ABB RAPID module: ReadTextMoveColor.mod

MODULE ReadTextMoveV2
    !   This module reads text from the target .txt file and moves to the points contained therein.
    !   Joshua Crook CM 1601   1-29-2016.
    VAR iodev pointsFile;
    PERS num paintHeight:=10;
    PERS num canvasHeight:=0;
    PERS num PAINT_MAX_DIST:=50;
    ! The largest usable square area the robot can draw in is 500mm wide by 150mm tall
    ! This is a rectangular large canvas, about 19.6" by 9.8"
    PERS num canvasXmin:=400;
    PERS num canvasXmax:=650;
    PERS num canvasYmin:=-250;
    PERS num canvasYmax:=250;

    VAR num sizeX;
    VAR num sizeY;
    VAR string tempStr;
    VAR num tempSF;
    VAR bool sizePassed:=FALSE;

    VAR num XTGT:=0;
    ! X target
    VAR num YTGT:=0;
    ! Y Target

    VAR num lastX:=0;
    VAR num lastY:=0;

    VAR string STRX;
    VAR string STRY;
    VAR string STRColor;
    VAR string lastColor:="A";
    !Arbitrary initialization value.

    VAR bool okX;
    VAR bool okY;
    VAR bool Skip;

    VAR num vX;
    VAR num vY;

    VAR num angleX;
    VAR num angleY;
    !measured in degrees from vertical.
    VAR num brushAngle:=10;

    VAR num vectorMag;
    VAR num distanceTravelled;

    PERS robtarget overA;
    PERS robtarget colorA;

    PERS robtarget overB;
    PERS robtarget colorB;

    PERS robtarget overC;
    PERS robtarget colorC;

    PERS robtarget overD;
    PERS robtarget colorD;

    PERS robtarget overE;
    PERS robtarget colorE;

    PERS robtarget overF;
    PERS robtarget colorF;

    PERS robtarget overClean;
    PERS robtarget clean;

    VAR num CaseHit;


    VAR orient ZeroZeroQuat:=[0.7071067811,0,0.7071067811,0];
    !vertical for paint can, etc.
    VAR orient paintStrokeQuat:=[0.7071067811,0,0.7071067811,0];
    !will change according to paintstroke vector.
    PERS num SF:=0.5;
    PERS num brushLength:=200;
    PERS num XOffset:=260;
    PERS num YOffset:=-150;
    PERS tooldata paintBrush:=[TRUE,[[87,0,146],[1,0,0,0]],[0.2,[0,0,146],[0,0,1,0],0,0,0]];

    PROC main()
        initializeColors;
        Open "HOME:/dumbSquare.txt",pointsFile\Read;
        distanceTravelled:=0;
        readSize;
        IF sizePassed=TRUE THEN
            readCoords;
            GotoPaint(STRColor);
            !first dip
            WHILE okX AND okY DO
                ! While we have data points in the file.
                moveToXY XTGT,YTGT;
                readCoords;
            ENDWHILE

        ENDIF

        Close pointsFile;
        ! exit.
    ENDPROC

    PROC initializeColors()
        overA:=[[514+brushLength,75,paintHeight+50],ZeroZeroQuat,[0,0,0,0],[9E9,9E9,9E9,9E9,9E9,9E9]];
        colorA:=[[514+brushLength,75,paintHeight],ZeroZeroQuat,[0,0,0,0],[9E9,9E9,9E9,9E9,9E9,9E9]];

        overB:=[[514+brushLength,50,paintHeight+50],ZeroZeroQuat,[0,0,0,0],[9E9,9E9,9E9,9E9,9E9,9E9]];
        colorB:=[[514+brushLength,50,paintHeight],ZeroZeroQuat,[0,0,0,0],[9E9,9E9,9E9,9E9,9E9,9E9]];

        overC:=[[514+brushLength,25,paintHeight+50],ZeroZeroQuat,[0,0,0,0],[9E9,9E9,9E9,9E9,9E9,9E9]];
        colorC:=[[514+brushLength,25,paintHeight],ZeroZeroQuat,[0,0,0,0],[9E9,9E9,9E9,9E9,9E9,9E9]];

        overD:=[[514+brushLength,0,paintHeight+50],ZeroZeroQuat,[0,0,0,0],[9E9,9E9,9E9,9E9,9E9,9E9]];
        colorD:=[[514+brushLength,0,paintHeight],ZeroZeroQuat,[0,0,0,0],[9E9,9E9,9E9,9E9,9E9,9E9]];

        overE:=[[514+brushLength,-25,paintHeight+50],ZeroZeroQuat,[0,0,0,0],[9E9,9E9,9E9,9E9,9E9,9E9]];
        colorE:=[[514+brushLength,-25,paintHeight],ZeroZeroQuat,[0,0,0,0],[9E9,9E9,9E9,9E9,9E9,9E9]];

        overF:=[[514+brushLength,-50,paintHeight+50],ZeroZeroQuat,[0,0,0,0],[9E9,9E9,9E9,9E9,9E9,9E9]];
        colorF:=[[514+brushLength,-50,paintHeight],ZeroZeroQuat,[0,0,0,0],[9E9,9E9,9E9,9E9,9E9,9E9]];

        overClean:=[[514+brushLength,-50,paintHeight+50],ZeroZeroQuat,[0,0,0,0],[9E9,9E9,9E9,9E9,9E9,9E9]];
        clean:=[[514+brushLength,-50,paintHeight],ZeroZeroQuat,[0,0,0,0],[9E9,9E9,9E9,9E9,9E9,9E9]];

    ENDPROC

    ! Reads the size off the passed file
    PROC readSize()
        sizePassed:=FALSE;
        ! This should be the X-size
        tempStr:=ReadStr(pointsFile\Delim:=",");
        okX:=StrToVal(tempStr,sizeX);
        ! This should be the Y-size
        tempStr:=ReadStr(pointsFile\Delim:=",");
        okY:=StrToVal(tempStr,sizeY);
        ! This should be a ';'
        tempStr:=ReadStr(pointsFile\Delim:=",");
        IF tempStr=";" THEN
            sizePassed:=TRUE;
            ! are we over the size constraints and in need of a scaling factor?
            IF (sizeX>(canvasXmax-canvasXmin)) OR (sizeY>(canvasYmax-canvasYmin)) THEN
                ! the Y proportion should be the scaling factor, as it was the smaller number
                IF ((canvasXmax-canvasXmin)/sizeX)>((canvasYmax-canvasYmin)/sizeY) THEN
                    SF:=(canvasYmax-canvasYmin)/sizeY;
                ELSE
                    SF:=(canvasXmax-canvasXmin)/sizeX;
                ENDIF

            ENDIF

        ELSE
            ErrLog 4800,"Data Error","The canvas size data was malformed","","","";
        ENDIF

    ENDPROC


    !   Reads the text file.
    PROC readCoords()
        STRX:=ReadStr(pointsFile\Delim:=",");
        okX:=StrToVal(STRX,XTGT);
        !End of a line.
        IF STRX=";" THEN
            STRColor:=ReadStr(pointsFile\Delim:=",");
            ! read the X value of the first point in the new line.
            STRX:=ReadStr(pointsFile\Delim:=",");
            STRY:=ReadStr(pointsFile\Delim:=",");

            okX:=StrToVal(STRX,XTGT);
            okY:=StrToVal(STRY,YTGT);

            checkForBadPoints XTGT,YTGT;

            XTGT:=(SF*XTGT)+canvasXmin;
            YTGT:=(SF*YTGT)+canvasYmin;
            CaseHit:=0;

        ELSEIF okX=FALSE THEN
            !Beginning of a file.
            STRColor:=STRX;
            STRX:=ReadStr(pointsFile\Delim:=",");
            STRY:=ReadStr(pointsFile\Delim:=",");

            okX:=StrToVal(STRX,XTGT);
            okY:=StrToVal(STRY,YTGT);

            checkForBadPoints XTGT,YTGT;

            XTGT:=(SF*XTGT)+canvasXmin;
            YTGT:=(SF*YTGT)+canvasYmin;
            lastX:=XTGT;
            lastY:=YTGT;
            CaseHit:=1;

        ELSEIF okX=TRUE THEN

            !we've already read the X value and it's not a character for a new line to be drawn.
            STRY:=ReadStr(pointsFile\Delim:=",");
            okY:=StrToVal(STRY,YTGT);

            checkForBadPoints XTGT,YTGT;

            XTGT:=(SF*XTGT)+canvasXmin;
            YTGT:=(SF*YTGT)+canvasYmin;
            CaseHit:=2;

        ENDIF
        !end of a file.
        IF (NOT okX) AND (NOT okY) THEN
            MoveL [[LastX,LastY,canvasHeight+30],ZeroZeroQuat,[0,0,0,0],[9E9,9E9,9E9,9E9,9E9,9E9]],v500,z0,paintBrush;
            MoveL overA,v500,fine,paintBrush;
        ENDIF
    ENDPROC

    ! Halts the robot if we get bad points.
    PROC checkForBadPoints(num Xcoord,num Ycoord)
        IF (Xcoord>sizeX) OR (Ycoord>sizeY) THEN
            ErrLog 4800,"Coord Error","One of the coordinates is outside expected bounds","Coordinates larger than image size are not allowed","-","-";
            TPWrite "Bad coordinates in the file: outside expected bounds";
            MoveL overA,v500,fine,paintBrush;
            Stop;
        ENDIF
        IF (Xcoord<0) OR (Ycoord<0) THEN
            ErrLog 4800,"Coord Error","Negative Coordinates are not allowed.","-","-","-";
            TPWrite "Bad coordinates in the file: outside expected bounds";
            MoveL overA,v500,fine,paintBrush;
            Stop;
        ENDIF

    ENDPROC

    PROC moveToXY(num XCoord,num YCoord)
        niceStroke;
        ConfL\Off;
        IF distanceTravelled>=PAINT_MAX_DIST OR CaseHit=0 THEN
            !if we've gone maximum distance or we reach the end of a line.
            GotoPaint(STRColor);
            distanceTravelled:=0;
        ENDIF
        IF NOT (CaseHit=0) THEN
            distanceTravelled:=distanceTravelled+vectorMag;
        ENDIF
        MoveL [[XCoord,YCoord,canvasHeight],paintStrokeQuat,[0,0,0,0],[9E9,9E9,9E9,9E9,9E9,9E9]],v100,z0,paintBrush;
        lastX:=XTGT;
        lastY:=YTGT;

        ! This moves to point at 100 mm/sec.
    ENDPROC

    PROC GotoPaint(string colorToPaint)
        !this is currently for blue paint only.
        ConfL\Off;
        !over target
        MoveL [[LastX,LastY,canvasHeight],paintStrokeQuat,[0,0,0,0],[9E9,9E9,9E9,9E9,9E9,9E9]],v100,fine,paintBrush;
        MoveL [[LastX,LastY,canvasHeight+30],ZeroZeroQuat,[0,0,0,0],[9E9,9E9,9E9,9E9,9E9,9E9]],v500,z0,paintBrush;
        IF (colorToPaint="A") THEN
            !over paint
            MoveL overA,v500,z0,paintBrush;
            !into paint
            MoveL colorA,v100,fine,paintBrush;
            !over paint
            MoveL overA,v500,z0,paintBrush;

        ELSEIF (colorToPaint="B") THEN
            !over paint
            MoveL overB,v500,z0,paintBrush;
            !into paint
            MoveL colorB,v100,fine,paintBrush;
            !over paint
            MoveL overB,v500,z0,paintBrush;
        ELSEIF (colorToPaint="C") THEN
            !over paint
            MoveL overC,v500,z0,paintBrush;
            !into paint
            MoveL colorC,v100,fine,paintBrush;
            !over paint
            MoveL overC,v500,z0,paintBrush;
        ELSEIF (colorToPaint="D") THEN
            !over paint
            MoveL overD,v500,z0,paintBrush;
            !into paint
            MoveL colorD,v100,fine,paintBrush;
            !over paint
            MoveL overD,v500,z0,paintBrush;
        ELSEIF (colorToPaint="E") THEN
            !over paint
            MoveL overE,v500,z0,paintBrush;
            !into paint
            MoveL colorE,v100,fine,paintBrush;
            !over paint
            MoveL overE,v500,z0,paintBrush;
        ELSEIF (colorToPaint="F") THEN
            !over paint
            MoveL overF,v500,z0,paintBrush;
            !into paint
            MoveL colorF,v100,fine,paintBrush;
            !over paint
            MoveL overF,v500,z0,paintBrush;

        ELSEIF (NOT (colorToPaint=lastColor)) THEN
            !NEED TO CLEAN
            MoveL overClean,v500,z0,paintBrush;
            MoveL clean,v100,fine,paintBrush;
            MoveL overClean,v500,z0,paintBrush;
        ENDIF
        !over target
        IF (CaseHit=0) THEN
            lastX:=XTGT;
            lastY:=YTGT;
        ENDIF
        MoveL [[LastX,LastY,canvasHeight+20],paintStrokeQuat,[0,0,0,0],[9E9,9E9,9E9,9E9,9E9,9E9]],v500,z0,paintBrush;
        MoveL [[LastX,LastY,canvasHeight],paintStrokeQuat,[0,0,0,0],[9E9,9E9,9E9,9E9,9E9,9E9]],v100,fine,paintBrush;
        lastColor:=colorToPaint;
    ENDPROC

    PROC niceStrokeQuat()
        !paintstroke vector
        vX:=XTGT-lastX;
        vY:=YTGT-lastY;
        vectorMag:=sqrt(vX*vX+vY*vY);

        angleY:=90+brushAngle;
        !Case to handle new lines.
        IF CaseHit=0 OR CaseHit=1 THEN
            paintStrokeQuat:=ZeroZeroQuat;

        ELSEIF vX>=0 AND vY>=0 THEN
            !PUSH
            paintStrokeQuat:=OrientZYX(ATan2(vY,vX),angleY,0);
        ELSEIF vX>=0 AND vY<=0 THEN
            !PUSH
            paintStrokeQuat:=OrientZYX(ATan2(vY,vX),angleY,0);
        ELSEIF vX<=0 AND vY>=0 THEN
            !PULL
            paintStrokeQuat:=OrientZYX(180-ATan2(vY,vX),180-angleY,0);
        ELSEIF vX<=0 AND vY<=0 THEN
            !PULL
            paintStrokeQuat:=OrientZYX(180-ATan2(vY,vX),angleY,0);
        ENDIF
    ENDPROC

    !   not really a nice stroke.
    PROC niceStroke()
        vX:=XTGT-lastX;
        vY:=YTGT-lastY;
        vectorMag:=sqrt(vX*vX+vY*vY);
        paintStrokeQuat:=ZeroZeroQuat;
    ENDPROC
ENDMODULE
